FUNCTION alg_g_algeb2: TupleStruct_1
VAR_INPUT
    state: STATE;
END_VAR


        alg_g_algeb2 := makeTupleStruct_1(state.curTime, (state.curTime) + (1.0));

END_FUNCTION

(* stored: ProductVersion 3.1.0.18, Version 1.1.0.1 *)
